  [665] = "-21.898000,-9.499000,118.777000,179.791000,0.392000,-123.893000,"
  [666] = "-21.901000,-9.495000,119.014000,179.790000,0.393000,-123.892000,"
  [667] = "-21.906000,-9.489000,119.373000,179.789000,0.396000,-123.892000,"
  [668] = "-21.912000,-9.481000,119.848000,179.788000,0.398000,-123.891000,"
  [669] = "-21.918000,-9.473000,120.297000,179.786000,0.401000,-123.890000,"
  [670] = "-21.923000,-9.467000,120.668000,179.785000,0.403000,-123.889000,"
  [671] = "-21.928000,-9.460000,121.039000,179.784000,0.406000,-123.888000,"
  [672] = "-21.845000,-9.093000,121.045000,179.788000,0.402000,-124.325000,"
  [673] = "-21.769000,-8.740000,121.052000,179.792000,0.397000,-124.728000,"
  [674] = "-21.697000,-8.391000,121.058000,179.797000,0.391000,-125.108000,"
  [675] = "-21.638000,-8.102000,121.063000,179.802000,0.385000,-125.409000,"
  [676] = "-21.575000,-7.782000,121.069000,179.807000,0.377000,-125.730000,"
  [677] = "-21.509000,-7.482000,121.076000,179.813000,0.367000,-126.051000,"
  [678] = "-21.413000,-7.146000,121.085000,179.824000,0.350000,-126.502000,"
  [679] = "-21.303000,-6.836000,121.095000,179.836000,0.330000,-127.021000,"
  [680] = "-21.191000,-6.564000,121.105000,179.848000,0.308000,-127.572000,"
  [681] = "-21.071000,-6.308000,121.115000,179.861000,0.286000,-128.189000,"
  [682] = "-20.932000,-6.069000,121.126000,179.875000,0.261000,-128.946000,"
  [683] = "-20.773000,-5.866000,121.138000,179.891000,0.232000,-129.864000,"
  [684] = "-20.590000,-5.697000,121.152000,179.909000,0.201000,-130.968000,"
  [685] = "-20.419000,-5.583000,121.164000,179.924000,0.172000,-132.053000,"
  [686] = "-20.230000,-5.492000,121.176000,179.939000,0.141000,-133.307000,"
  [687] = "-20.054000,-5.404000,121.187000,179.952000,0.115000,-134.556000,"
  [688] = "-19.877000,-5.305000,121.198000,179.963000,0.093000,-135.914000,"
  [689] = "-19.712000,-5.201000,121.207000,179.971000,0.074000,-137.273000,"
  [690] = "-19.569000,-5.104000,121.215000,179.977000,0.061000,-138.523000,"
  [691] = "-19.444000,-5.013000,121.222000,179.982000,0.050000,-139.689000,"
  [692] = "-19.298000,-4.901000,121.230000,179.986000,0.040000,-141.114000,"
  [693] = "-19.179000,-4.805000,121.236000,179.989000,0.033000,-142.336000,"
  [694] = "-19.074000,-4.717000,121.241000,179.991000,0.028000,-143.461000,"
  [695] = "-18.958000,-4.618000,121.246000,179.993000,0.023000,-144.749000,"
  [696] = "-18.847000,-4.521000,121.251000,179.994000,0.019000,-146.026000,"
  [697] = "-18.726000,-4.408000,121.257000,179.995000,0.015000,-147.486000,"
  [698] = "-18.617000,-4.297000,121.262000,179.996000,0.014000,-148.881000,"
  [699] = "-18.518000,-4.187000,121.266000,179.996000,0.014000,-150.220000,"
  [700] = "-18.428000,-4.079000,121.269000,179.996000,0.015000,-151.511000,"
  [701] = "-18.346000,-3.973000,121.272000,179.996000,0.018000,-152.759000,"
  [702] = "-18.250000,-3.838000,121.276000,179.995000,0.023000,-154.311000,"
  [703] = "-18.184000,-3.736000,121.278000,179.994000,0.029000,-155.473000,"
  [704] = "-18.124000,-3.635000,121.280000,179.993000,0.035000,-156.607000,"
  [705] = "-18.070000,-3.536000,121.281000,179.992000,0.042000,-157.716000,"
  [706] = "-17.998000,-3.393000,121.282000,179.990000,0.054000,-159.311000,"
  [707] = "-17.935000,-3.250000,121.283000,179.989000,0.068000,-160.916000,"
  [708] = "-17.880000,-3.116000,121.283000,179.987000,0.083000,-162.465000,"
  [709] = "-17.832000,-2.989000,121.283000,179.986000,0.099000,-163.999000,"
  [710] = "-17.789000,-2.868000,121.283000,179.985000,0.116000,-165.512000,"
  [711] = "-17.752000,-2.754000,121.282000,179.985000,0.134000,-167.010000,"
  [712] = "-17.720000,-2.646000,121.280000,179.985000,0.152000,-168.496000,"
  [713] = "-17.692000,-2.545000,121.279000,179.985000,0.171000,-169.972000,"
  [714] = "-17.668000,-2.449000,121.277000,179.986000,0.190000,-171.441000,"
  [715] = "-17.648000,-2.360000,121.275000,179.987000,0.210000,-172.903000,"
  [716] = "-17.631000,-2.277000,121.272000,179.989000,0.230000,-174.360000,"
  [717] = "-17.618000,-2.198000,121.269000,179.991000,0.251000,-175.808000,"
  [718] = "-17.612000,-2.118000,121.266000,179.993000,0.274000,-177.225000,"
  [719] = "-17.612000,-2.038000,121.262000,179.996000,0.298000,-178.614000,"
  [720] = "-17.621000,-1.930000,121.257000,-179.999000,0.331000,179.575000,"
  [721] = "-17.638000,-1.823000,121.250000,-179.993000,0.367000,177.803000,"
  [722] = "-17.664000,-1.717000,121.244000,-179.986000,0.404000,176.064000,"
  [723] = "-17.695000,-1.613000,121.236000,-179.978000,0.442000,174.351000,"
  [724] = "-17.729000,-1.512000,121.229000,-179.969000,0.479000,172.658000,"
  [725] = "-17.763000,-1.413000,121.222000,-179.959000,0.514000,170.982000,"
  [726] = "-17.796000,-1.317000,121.215000,-179.949000,0.547000,169.318000,"
  [727] = "-17.826000,-1.220000,121.209000,-179.938000,0.577000,167.683000,"
  [728] = "-17.857000,-1.115000,121.203000,-179.926000,0.605000,166.103000,"
  [729] = "-17.891000,-1.003000,121.197000,-179.914000,0.632000,164.577000,"
  [730] = "-17.927000,-0.883000,121.191000,-179.902000,0.658000,163.102000,"
  [731] = "-17.966000,-0.756000,121.185000,-179.890000,0.684000,161.676000,"
  [732] = "-18.010000,-0.622000,121.179000,-179.877000,0.710000,160.296000,"
  [733] = "-18.058000,-0.482000,121.172000,-179.863000,0.736000,158.960000,"
  [734] = "-18.112000,-0.336000,121.166000,-179.850000,0.762000,157.664000,"
  [735] = "-18.171000,-0.184000,121.159000,-179.835000,0.789000,156.408000,"
  [736] = "-18.236000,-0.028000,121.152000,-179.820000,0.817000,155.188000,"
  [737] = "-18.306000,0.130000,121.144000,-179.805000,0.846000,153.987000,"
  [738] = "-18.381000,0.285000,121.137000,-179.788000,0.875000,152.777000,"
  [739] = "-18.458000,0.435000,121.129000,-179.771000,0.903000,151.558000,"
  [740] = "-18.540000,0.581000,121.121000,-179.753000,0.932000,150.327000,"
  [741] = "-18.624000,0.723000,121.114000,-179.735000,0.959000,149.084000,"
  [742] = "-18.712000,0.860000,121.106000,-179.715000,0.987000,147.828000,"
  [743] = "-18.803000,0.992000,121.098000,-179.695000,1.014000,146.557000,"
  [744] = "-18.898000,1.119000,121.090000,-179.675000,1.040000,145.269000,"
  [745] = "-18.995000,1.242000,121.082000,-179.653000,1.066000,143.964000,"
  [746] = "-19.096000,1.359000,121.074000,-179.631000,1.091000,142.641000,"
  [747] = "-19.201000,1.474000,121.066000,-179.608000,1.116000,141.314000,"
  [748] = "-19.311000,1.597000,121.057000,-179.584000,1.143000,140.029000,"
  [749] = "-19.426000,1.728000,121.048000,-179.560000,1.171000,138.787000,"
  [750] = "-19.515000,1.831000,121.041000,-179.541000,1.193000,137.884000,"
  [751] = "-19.636000,1.977000,121.032000,-179.515000,1.222000,136.718000,"
  [752] = "-19.760000,2.132000,121.023000,-179.489000,1.252000,135.595000,"
  [753] = "-19.886000,2.297000,121.013000,-179.463000,1.282000,134.516000,"
  [754] = "-20.012000,2.472000,121.004000,-179.436000,1.312000,133.480000,"
  [755] = "-20.139000,2.659000,120.995000,-179.410000,1.341000,132.487000,"
  [756] = "-20.266000,2.856000,120.986000,-179.384000,1.369000,131.536000,"
  [757] = "-20.384000,3.053000,120.978000,-179.360000,1.394000,130.664000,"
  [758] = "-20.507000,3.265000,120.970000,-179.335000,1.418000,129.754000,"
  [759] = "-20.629000,3.481000,120.963000,-179.311000,1.440000,128.848000,"
  [760] = "-20.750000,3.700000,120.956000,-179.287000,1.460000,127.946000,"
  [761] = "-20.872000,3.924000,120.950000,-179.264000,1.478000,127.048000,"
  [762] = "-20.996000,4.150000,120.944000,-179.241000,1.495000,126.155000,"
  [763] = "-21.122000,4.379000,120.938000,-179.217000,1.512000,125.265000,"
  [764] = "-21.251000,4.611000,120.932000,-179.194000,1.528000,124.379000,"
  [765] = "-21.384000,4.845000,120.926000,-179.170000,1.544000,123.496000,"
  [766] = "-21.523000,5.081000,120.920000,-179.146000,1.560000,122.619000,"
  [767] = "-21.664000,5.325000,120.914000,-179.121000,1.579000,121.783000,"
  [768] = "-21.804000,5.576000,120.908000,-179.096000,1.598000,121.012000,"
  [769] = "-21.925000,5.801000,120.902000,-179.074000,1.616000,120.389000,"
  [770] = "-22.025000,5.996000,120.898000,-179.056000,1.632000,119.897000,"
  [771] = "-22.164000,6.281000,120.892000,-179.030000,1.654000,119.251000,"
  [772] = "-22.281000,6.538000,120.887000,-179.009000,1.674000,118.737000,"
  [773] = "-22.383000,6.779000,120.883000,-178.990000,1.691000,118.306000,"
  [774] = "-22.481000,7.031000,120.879000,-178.972000,1.708000,117.907000,"
  [775] = "-22.565000,7.263000,120.876000,-178.957000,1.722000,117.578000,"
  [776] = "-22.664000,7.566000,120.873000,-178.938000,1.739000,117.202000,"
  [777] = "-22.739000,7.817000,120.871000,-178.925000,1.752000,116.922000,"
  [778] = "-22.828000,8.137000,120.869000,-178.909000,1.765000,116.585000,"
  [779] = "-22.896000,8.399000,120.868000,-178.898000,1.775000,116.326000,"
  [780] = "-22.977000,8.733000,120.867000,-178.885000,1.785000,116.016000,"
  [781] = "-23.040000,9.006000,120.866000,-178.875000,1.793000,115.779000,"
  [782] = "-23.114000,9.353000,120.866000,-178.863000,1.801000,115.496000,"
  [783] = "-23.172000,9.636000,120.867000,-178.855000,1.807000,115.281000,"
  [784] = "-23.241000,9.995000,120.867000,-178.845000,1.814000,115.026000,"
  [785] = "-23.295000,10.287000,120.868000,-178.837000,1.820000,114.833000,"
  [786] = "-23.360000,10.657000,120.868000,-178.827000,1.827000,114.607000,"
  [787] = "-23.411000,10.956000,120.869000,-178.820000,1.832000,114.438000,"
  [788] = "-23.475000,11.334000,120.870000,-178.811000,1.840000,114.235000,"
  [789] = "-23.528000,11.637000,120.871000,-178.803000,1.846000,114.071000,"
  [790] = "-23.595000,12.015000,120.873000,-178.793000,1.853000,113.864000,"
  [791] = "-23.657000,12.356000,120.874000,-178.785000,1.859000,113.675000,"
  [792] = "-23.720000,12.697000,120.875000,-178.776000,1.866000,113.485000,"
  [793] = "-23.785000,13.039000,120.876000,-178.768000,1.872000,113.292000,"
  [794] = "-23.852000,13.381000,120.878000,-178.759000,1.878000,113.098000,"
  [795] = "-23.920000,13.723000,120.879000,-178.751000,1.884000,112.902000,"
  [796] = "-23.989000,14.066000,120.880000,-178.742000,1.890000,112.703000,"
  [797] = "-24.060000,14.410000,120.882000,-178.734000,1.895000,112.503000,"
  [798] = "-24.132000,14.754000,120.884000,-178.725000,1.901000,112.300000,"
  [799] = "-24.205000,15.098000,120.885000,-178.717000,1.906000,112.095000,"
  [800] = "-24.280000,15.443000,120.887000,-178.709000,1.910000,111.888000,"
  [801] = "-24.357000,15.789000,120.889000,-178.701000,1.915000,111.679000,"
  [802] = "-24.434000,16.135000,120.891000,-178.693000,1.919000,111.468000,"
  [803] = "-24.504000,16.444000,120.893000,-178.686000,1.922000,111.278000,"
  [804] = "-24.593000,16.831000,120.895000,-178.677000,1.926000,111.038000,"
  [805] = "-24.666000,17.141000,120.897000,-178.671000,1.929000,110.844000,"
  [806] = "-24.758000,17.529000,120.899000,-178.663000,1.931000,110.599000,"
  [807] = "-24.833000,17.841000,120.901000,-178.656000,1.933000,110.401000,"
  [808] = "-24.928000,18.232000,120.904000,-178.649000,1.935000,110.151000,"
  [809] = "-25.004000,18.546000,120.906000,-178.643000,1.936000,109.950000,"
  [810] = "-25.099000,18.941000,120.909000,-178.636000,1.937000,109.702000,"
  [811] = "-25.175000,19.259000,120.911000,-178.631000,1.938000,109.507000,"
  [812] = "-25.270000,19.660000,120.914000,-178.624000,1.938000,109.268000,"
  [813] = "-25.347000,19.982000,120.917000,-178.619000,1.939000,109.079000,"
  [814] = "-25.442000,20.388000,120.920000,-178.612000,1.940000,108.847000,"
  [815] = "-25.519000,20.713000,120.923000,-178.607000,1.941000,108.665000,"
  [816] = "-25.616000,21.122000,120.926000,-178.599000,1.943000,108.442000,"
  [817] = "-25.695000,21.451000,120.928000,-178.593000,1.945000,108.267000,"
  [818] = "-25.795000,21.863000,120.932000,-178.585000,1.949000,108.052000,"
  [819] = "-25.876000,22.194000,120.934000,-178.578000,1.953000,107.883000,"
  [820] = "-25.980000,22.607000,120.938000,-178.569000,1.957000,107.673000,"
  [821] = "-26.063000,22.939000,120.941000,-178.562000,1.961000,107.505000,"
  [822] = "-26.167000,23.357000,120.944000,-178.553000,1.966000,107.296000,"
  [823] = "-26.266000,23.765000,120.948000,-178.546000,1.968000,107.095000,"
  [824] = "-26.349000,24.120000,120.951000,-178.541000,1.969000,106.922000,"
  [825] = "-26.440000,24.538000,120.955000,-178.537000,1.967000,106.722000,"
  [826] = "-26.514000,24.903000,120.959000,-178.536000,1.962000,106.550000,"
  [827] = "-26.587000,25.305000,120.963000,-178.537000,1.954000,106.365000,"
  [828] = "-26.667000,25.705000,120.967000,-178.542000,1.940000,106.150000,"
  [829] = "-26.663000,25.706000,121.384000,-178.542000,1.941000,106.158000,"
  [830] = "-26.659000,25.708000,121.801000,-178.542000,1.941000,106.166000,"
  [831] = "-26.656000,25.710000,122.168000,-178.542000,1.941000,106.174000,"
  [832] = "-26.652000,25.711000,122.585000,-178.542000,1.941000,106.182000,"
  [833] = "-26.649000,25.713000,122.951000,-178.542000,1.941000,106.189000,"
  [834] = "-26.645000,25.714000,123.369000,-178.542000,1.941000,106.198000,"
  [835] = "-26.640000,25.716000,123.843000,-178.542000,1.941000,106.207000,"
  [836] = "-26.636000,25.718000,124.292000,-178.543000,1.942000,106.216000,"
  [837] = "-26.633000,25.719000,124.657000,-178.543000,1.942000,106.223000,"
  [838] = "-26.629000,25.721000,125.023000,-178.543000,1.942000,106.231000,"
  [839] = "-26.566000,25.344000,125.019000,-178.537000,1.956000,106.418000,"
  [840] = "-26.510000,24.896000,125.015000,-178.534000,1.966000,106.575000,"
  [841] = "-26.451000,24.520000,125.011000,-178.534000,1.970000,106.716000,"
  [842] = "-26.372000,24.093000,125.006000,-178.538000,1.972000,106.887000,"
  [843] = "-26.297000,23.732000,125.003000,-178.543000,1.971000,107.040000,"
  [844] = "-26.203000,23.321000,124.999000,-178.550000,1.967000,107.225000,"
  [845] = "-26.101000,22.902000,124.995000,-178.560000,1.962000,107.424000,"
  [846] = "-26.016000,22.570000,124.992000,-178.567000,1.957000,107.588000,"
  [847] = "-25.909000,22.159000,124.989000,-178.577000,1.951000,107.802000,"
  [848] = "-25.824000,21.831000,124.987000,-178.585000,1.947000,107.977000,"
  [849] = "-25.720000,21.422000,124.983000,-178.593000,1.944000,108.201000,"
  [850] = "-25.639000,21.096000,124.981000,-178.599000,1.942000,108.382000,"
  [851] = "-25.539000,20.688000,124.978000,-178.606000,1.940000,108.611000,"
  [852] = "-25.462000,20.363000,124.975000,-178.611000,1.939000,108.796000,"
  [853] = "-25.366000,19.958000,124.972000,-178.618000,1.939000,109.030000,"
  [854] = "-25.290000,19.635000,124.969000,-178.623000,1.939000,109.220000,"
  [855] = "-25.196000,19.234000,124.966000,-178.629000,1.939000,109.459000,"
  [856] = "-25.122000,18.914000,124.964000,-178.634000,1.938000,109.652000,"
  [857] = "-25.028000,18.518000,124.961000,-178.640000,1.938000,109.896000,"
  [858] = "-24.953000,18.202000,124.959000,-178.646000,1.937000,110.093000,"
  [859] = "-24.860000,17.810000,124.956000,-178.653000,1.936000,110.338000,"
  [860] = "-24.787000,17.497000,124.954000,-178.659000,1.934000,110.533000,"
  [861] = "-24.696000,17.107000,124.951000,-178.667000,1.931000,110.773000,"
  [862] = "-24.624000,16.796000,124.949000,-178.674000,1.928000,110.963000,"
  [863] = "-24.535000,16.409000,124.947000,-178.682000,1.924000,111.199000,"
  [864] = "-24.465000,16.100000,124.945000,-178.689000,1.921000,111.386000,"
  [865] = "-24.379000,15.714000,124.943000,-178.698000,1.916000,111.617000,"
  [866] = "-24.311000,15.407000,124.941000,-178.706000,1.912000,111.800000,"
  [867] = "-24.228000,15.023000,124.939000,-178.715000,1.906000,112.027000,"
  [868] = "-24.162000,14.717000,124.938000,-178.723000,1.901000,112.207000,"
  [869] = "-24.081000,14.335000,124.936000,-178.732000,1.895000,112.430000,"
  [870] = "-24.018000,14.030000,124.935000,-178.740000,1.890000,112.606000,"
  [871] = "-23.940000,13.649000,124.933000,-178.749000,1.883000,112.825000,"
  [872] = "-23.879000,13.345000,124.932000,-178.757000,1.878000,112.998000,"
  [873] = "-23.804000,12.965000,124.930000,-178.767000,1.871000,113.213000,"
  [874] = "-23.746000,12.662000,124.929000,-178.775000,1.865000,113.383000,"
  [875] = "-23.674000,12.283000,124.928000,-178.784000,1.858000,113.594000,"
  [876] = "-23.618000,11.980000,124.927000,-178.792000,1.852000,113.761000,"
  [877] = "-23.550000,11.602000,124.926000,-178.802000,1.844000,113.969000,"
  [878] = "-23.497000,11.300000,124.925000,-178.809000,1.838000,114.133000,"
  [879] = "-23.433000,10.923000,124.924000,-178.818000,1.831000,114.337000,"
  [880] = "-23.381000,10.623000,124.923000,-178.826000,1.826000,114.507000,"
  [881] = "-23.315000,10.253000,124.922000,-178.835000,1.819000,114.731000,"
  [882] = "-23.262000,9.960000,124.921000,-178.843000,1.813000,114.920000,"
  [883] = "-23.193000,9.599000,124.921000,-178.853000,1.806000,115.168000,"
  [884] = "-23.136000,9.315000,124.921000,-178.861000,1.800000,115.376000,"
  [885] = "-23.063000,8.965000,124.921000,-178.873000,1.792000,115.648000,"
  [886] = "-23.002000,8.689000,124.921000,-178.883000,1.784000,115.874000,"
  [887] = "-22.922000,8.351000,124.922000,-178.896000,1.773000,116.168000,"
  [888] = "-22.855000,8.085000,124.923000,-178.907000,1.763000,116.411000,"
  [889] = "-22.767000,7.760000,124.925000,-178.923000,1.749000,116.727000,"
  [890] = "-22.693000,7.505000,124.927000,-178.936000,1.736000,116.989000,"
  [891] = "-22.595000,7.198000,124.930000,-178.954000,1.718000,117.348000,"
  [892] = "-22.511000,6.963000,124.933000,-178.970000,1.703000,117.665000,"
  [893] = "-22.401000,6.681000,124.937000,-178.990000,1.685000,118.100000,"
  [894] = "-22.268000,6.370000,124.943000,-179.014000,1.662000,118.660000,"
  [895] = "-22.169000,6.158000,124.947000,-179.032000,1.646000,119.094000,"
  [896] = "-22.049000,5.914000,124.952000,-179.054000,1.627000,119.652000,"
  [897] = "-21.908000,5.644000,124.958000,-179.079000,1.606000,120.352000,"
  [898] = "-21.763000,5.382000,124.964000,-179.105000,1.586000,121.122000,"
  [899] = "-21.619000,5.133000,124.971000,-179.130000,1.567000,121.949000,"
  [900] = "-21.477000,4.896000,124.977000,-179.155000,1.550000,122.824000,"
  [901] = "-21.340000,4.662000,124.983000,-179.179000,1.534000,123.711000,"
  [902] = "-21.208000,4.430000,124.988000,-179.203000,1.518000,124.596000,"
  [903] = "-21.078000,4.199000,124.994000,-179.226000,1.502000,125.482000,"
  [904] = "-20.952000,3.971000,125.001000,-179.250000,1.485000,126.368000,"
  [905] = "-20.827000,3.745000,125.007000,-179.273000,1.466000,127.255000,"
  [906] = "-20.703000,3.521000,125.014000,-179.297000,1.446000,128.142000,"
  [907] = "-20.580000,3.301000,125.021000,-179.321000,1.424000,129.030000,"
  [908] = "-20.455000,3.084000,125.029000,-179.346000,1.400000,129.920000,"
  [909] = "-20.329000,2.870000,125.037000,-179.371000,1.374000,130.811000,"
  [910] = "-20.208000,2.676000,125.045000,-179.396000,1.347000,131.684000,"
  [911] = "-20.080000,2.483000,125.054000,-179.422000,1.318000,132.648000,"
  [912] = "-19.952000,2.301000,125.064000,-179.448000,1.289000,133.658000,"
  [913] = "-19.824000,2.131000,125.073000,-179.475000,1.259000,134.714000,"
  [914] = "-19.699000,1.972000,125.082000,-179.501000,1.230000,135.817000,"
  [915] = "-19.576000,1.822000,125.092000,-179.527000,1.200000,136.966000,"
  [916] = "-19.457000,1.682000,125.101000,-179.552000,1.172000,138.161000,"
  [917] = "-19.399000,1.616000,125.105000,-179.564000,1.158000,138.777000,"
  [918] = "-19.285000,1.490000,125.114000,-179.589000,1.131000,140.042000,"
  [919] = "-19.176000,1.373000,125.122000,-179.612000,1.106000,141.353000,"
  [920] = "-19.072000,1.259000,125.130000,-179.635000,1.081000,142.688000,"
  [921] = "-18.971000,1.141000,125.138000,-179.657000,1.055000,144.005000,"
  [922] = "-18.872000,1.018000,125.146000,-179.679000,1.029000,145.304000,"
  [923] = "-18.777000,0.889000,125.154000,-179.699000,1.002000,146.586000,"
  [924] = "-18.684000,0.756000,125.163000,-179.719000,0.974000,147.852000,"
  [925] = "-18.595000,0.619000,125.170000,-179.739000,0.946000,149.104000,"
  [926] = "-18.510000,0.477000,125.178000,-179.757000,0.918000,150.343000,"
  [927] = "-18.427000,0.330000,125.186000,-179.775000,0.889000,151.571000,"
  [928] = "-18.349000,0.180000,125.194000,-179.792000,0.861000,152.788000,"
  [929] = "-18.275000,0.026000,125.201000,-179.808000,0.832000,153.997000,"
  [930] = "-18.205000,-0.131000,125.209000,-179.823000,0.803000,155.207000,"
  [931] = "-18.142000,-0.284000,125.216000,-179.838000,0.776000,156.448000,"
  [932] = "-18.086000,-0.432000,125.222000,-179.852000,0.750000,157.723000,"
  [933] = "-18.034000,-0.574000,125.229000,-179.866000,0.724000,159.035000,"
  [934] = "-17.987000,-0.712000,125.235000,-179.879000,0.699000,160.385000,"
  [935] = "-17.945000,-0.843000,125.241000,-179.892000,0.674000,161.777000,"
  [936] = "-17.906000,-0.968000,125.247000,-179.904000,0.648000,163.212000,"
  [937] = "-17.869000,-1.087000,125.253000,-179.917000,0.621000,164.692000,"
  [938] = "-17.834000,-1.199000,125.259000,-179.928000,0.593000,166.221000,"
  [939] = "-17.800000,-1.304000,125.266000,-179.940000,0.564000,167.801000,"
  [940] = "-17.765000,-1.404000,125.272000,-179.951000,0.532000,169.423000,"
  [941] = "-17.727000,-1.504000,125.280000,-179.961000,0.497000,171.067000,"
  [942] = "-17.690000,-1.605000,125.287000,-179.971000,0.460000,172.733000,"
  [943] = "-17.655000,-1.707000,125.295000,-179.979000,0.422000,174.427000,"
  [944] = "-17.625000,-1.809000,125.302000,-179.987000,0.385000,176.153000,"
  [945] = "-17.604000,-1.911000,125.308000,-179.994000,0.349000,177.913000,"
  [946] = "-17.591000,-2.014000,125.314000,-179.999000,0.315000,179.710000,"
  [947] = "-17.588000,-2.116000,125.319000,179.996000,0.284000,-178.451000,"
  [948] = "-17.593000,-2.192000,125.322000,179.993000,0.261000,-177.039000,"
  [949] = "-17.604000,-2.267000,125.325000,179.991000,0.241000,-175.597000,"
  [950] = "-17.619000,-2.345000,125.328000,179.989000,0.221000,-174.138000,"
  [951] = "-17.638000,-2.428000,125.330000,179.987000,0.201000,-172.675000,"
  [952] = "-17.660000,-2.517000,125.332000,179.986000,0.182000,-171.208000,"
  [953] = "-17.686000,-2.612000,125.334000,179.985000,0.163000,-169.733000,"
  [954] = "-17.716000,-2.713000,125.335000,179.985000,0.145000,-168.250000,"
  [955] = "-17.750000,-2.820000,125.336000,179.985000,0.127000,-166.757000,"
  [956] = "-17.789000,-2.934000,125.337000,179.986000,0.110000,-165.250000,"
  [957] = "-17.833000,-3.054000,125.338000,179.987000,0.093000,-163.727000,"
  [958] = "-17.883000,-3.181000,125.338000,179.988000,0.078000,-162.184000,"
  [959] = "-17.940000,-3.312000,125.337000,179.989000,0.063000,-160.636000,"
  [960] = "-18.006000,-3.452000,125.337000,179.991000,0.050000,-159.018000,"
  [961] = "-18.081000,-3.589000,125.335000,179.992000,0.038000,-157.421000,"
  [962] = "-18.137000,-3.685000,125.333000,179.993000,0.032000,-156.307000,"
  [963] = "-18.199000,-3.782000,125.332000,179.994000,0.026000,-155.167000,"
  [964] = "-18.267000,-3.880000,125.329000,179.995000,0.022000,-153.999000,"
  [965] = "-18.365000,-4.010000,125.326000,179.996000,0.017000,-152.435000,"
  [966] = "-18.450000,-4.112000,125.323000,179.996000,0.015000,-151.181000,"
  [967] = "-18.542000,-4.216000,125.319000,179.996000,0.014000,-149.885000,"
  [968] = "-18.643000,-4.321000,125.315000,179.996000,0.014000,-148.540000,"
  [969] = "-18.755000,-4.427000,125.310000,179.995000,0.016000,-147.139000,"
  [970] = "-18.878000,-4.535000,125.304000,179.994000,0.020000,-145.674000,"
  [971] = "-19.010000,-4.645000,125.298000,179.992000,0.025000,-144.177000,"
  [972] = "-19.107000,-4.723000,125.294000,179.990000,0.030000,-143.115000,"
  [973] = "-19.218000,-4.808000,125.288000,179.987000,0.036000,-141.964000,"
  [974] = "-19.354000,-4.908000,125.281000,179.984000,0.046000,-140.605000,"
  [975] = "-19.499000,-5.005000,125.273000,179.979000,0.058000,-139.248000,"
  [976] = "-19.654000,-5.101000,125.265000,179.972000,0.073000,-137.874000,"
  [977] = "-19.807000,-5.186000,125.256000,179.964000,0.090000,-136.608000,"
  [978] = "-19.967000,-5.265000,125.247000,179.955000,0.110000,-135.363000,"
  [979] = "-20.149000,-5.343000,125.235000,179.942000,0.136000,-134.032000,"
  [980] = "-20.364000,-5.424000,125.222000,179.925000,0.170000,-132.579000,"
  [981] = "-20.532000,-5.511000,125.210000,179.911000,0.198000,-131.491000,"
  [982] = "-20.715000,-5.648000,125.197000,179.894000,0.229000,-130.351000,"
  [983] = "-20.882000,-5.823000,125.185000,179.878000,0.258000,-129.365000,"
  [984] = "-21.030000,-6.037000,125.173000,179.863000,0.285000,-128.524000,"
  [985] = "-21.152000,-6.267000,125.163000,179.850000,0.307000,-127.874000,"
  [986] = "-21.267000,-6.517000,125.153000,179.837000,0.328000,-127.293000,"
  [987] = "-21.382000,-6.815000,125.143000,179.825000,0.350000,-126.739000,"
  [988] = "-21.480000,-7.132000,125.134000,179.814000,0.367000,-126.276000,"
  [989] = "-21.543000,-7.396000,125.128000,179.807000,0.378000,-125.972000,"
  [990] = "-21.598000,-7.692000,125.122000,179.802000,0.385000,-125.695000,"
  [991] = "-21.665000,-8.058000,125.116000,179.797000,0.393000,-125.347000,"
  [992] = "-21.733000,-8.421000,125.109000,179.792000,0.399000,-124.984000,"
  [993] = "-21.787000,-8.696000,125.105000,179.789000,0.403000,-124.695000,"
  [994] = "-21.858000,-9.046000,125.099000,179.785000,0.407000,-124.311000,"
  [995] = "-21.936000,-9.408000,125.093000,179.782000,0.410000,-123.894000,"
  [996] = "-21.933000,-9.407000,125.510000,179.782000,0.408000,-123.892000,"
  [997] = "-21.930000,-9.405000,125.928000,179.783000,0.407000,-123.891000,"
  [998] = "-21.927000,-9.404000,126.295000,179.784000,0.405000,-123.890000,"
  [999] = "-21.924000,-9.403000,126.712000,179.785000,0.404000,-123.888000,"
  [1000] = "-21.921000,-9.402000,127.079000,179.785000,0.403000,-123.887000,"
  [1001] = "-21.918000,-9.401000,127.497000,179.786000,0.401000,-123.886000,"
  [1002] = "-21.914000,-9.399000,127.970000,179.787000,0.399000,-123.884000,"
  [1003] = "-21.911000,-9.398000,128.420000,179.788000,0.398000,-123.882000,"
  [1004] = "-21.908000,-9.397000,128.785000,179.789000,0.396000,-123.881000,"
  [1005] = "-21.905000,-9.396000,129.151000,179.789000,0.395000,-123.880000,"
  [1006] = "-21.841000,-9.094000,129.156000,179.792000,0.392000,-124.222000,"
  [1007] = "-21.767000,-8.722000,129.162000,179.796000,0.389000,-124.623000,"
  [1008] = "-21.698000,-8.350000,129.168000,179.800000,0.384000,-125.001000,"
  [1009] = "-21.636000,-7.996000,129.174000,179.804000,0.379000,-125.341000,"
  [1010] = "-21.574000,-7.627000,129.180000,179.808000,0.373000,-125.674000,"
  [1011] = "-21.527000,-7.331000,129.186000,179.812000,0.368000,-125.928000,"
  [1012] = "-21.474000,-7.055000,129.191000,179.817000,0.360000,-126.199000,"
  [1013] = "-21.387000,-6.733000,129.199000,179.826000,0.346000,-126.623000,"
  [1014] = "-21.274000,-6.415000,129.210000,179.838000,0.326000,-127.185000,"
  [1015] = "-21.178000,-6.199000,129.218000,179.848000,0.308000,-127.673000,"
  [1016] = "-21.058000,-5.968000,129.228000,179.861000,0.287000,-128.317000,"
  [1017] = "-20.945000,-5.787000,129.236000,179.872000,0.268000,-128.961000,"
  [1018] = "-20.800000,-5.610000,129.247000,179.886000,0.243000,-129.828000,"
  [1019] = "-20.652000,-5.478000,129.258000,179.900000,0.219000,-130.741000,"
  [1020] = "-20.476000,-5.365000,129.270000,179.915000,0.190000,-131.877000,"
  [1021] = "-20.289000,-5.287000,129.282000,179.931000,0.160000,-133.120000,"
  [1022] = "-20.088000,-5.227000,129.295000,179.946000,0.129000,-134.508000,"
  [1023] = "-19.895000,-5.156000,129.306000,179.959000,0.102000,-135.941000,"
  [1024] = "-19.715000,-5.077000,129.317000,179.969000,0.080000,-137.368000,"
  [1025] = "-19.561000,-4.999000,129.326000,179.976000,0.063000,-138.682000,"
  [1026] = "-19.427000,-4.922000,129.333000,179.982000,0.050000,-139.885000,"
  [1027] = "-19.274000,-4.826000,129.341000,179.987000,0.038000,-141.341000,"
  [1028] = "-19.151000,-4.740000,129.347000,179.990000,0.030000,-142.591000,"
  [1029] = "-19.043000,-4.661000,129.352000,179.992000,0.024000,-143.734000,"
  [1030] = "-18.902000,-4.550000,129.359000,179.994000,0.018000,-145.305000,"
  [1031] = "-18.775000,-4.444000,129.365000,179.996000,0.014000,-146.807000,"
  [1032] = "-18.658000,-4.341000,129.370000,179.997000,0.011000,-148.246000,"
  [1033] = "-18.553000,-4.238000,129.374000,179.997000,0.010000,-149.624000,"
  [1034] = "-18.457000,-4.137000,129.378000,179.997000,0.011000,-150.951000,"
  [1035] = "-18.370000,-4.037000,129.381000,179.997000,0.012000,-152.231000,"
  [1036] = "-18.290000,-3.938000,129.384000,179.996000,0.015000,-153.473000,"
  [1037] = "-18.217000,-3.841000,129.387000,179.996000,0.020000,-154.679000,"
  [1038] = "-18.151000,-3.745000,129.389000,179.995000,0.025000,-155.853000,"
  [1039] = "-18.090000,-3.651000,129.390000,179.994000,0.031000,-157.000000,"
  [1040] = "-18.035000,-3.558000,129.392000,179.993000,0.038000,-158.121000,"
  [1041] = "-17.962000,-3.424000,129.393000,179.991000,0.049000,-159.732000,"
  [1042] = "-17.898000,-3.289000,129.394000,179.990000,0.063000,-161.357000,"
  [1043] = "-17.843000,-3.162000,129.394000,179.988000,0.078000,-162.916000,"
  [1044] = "-17.795000,-3.040000,129.394000,179.987000,0.094000,-164.461000,"
  [1045] = "-17.752000,-2.925000,129.393000,179.986000,0.111000,-165.983000,"
  [1046] = "-17.715000,-2.816000,129.392000,179.986000,0.128000,-167.488000,"
  [1047] = "-17.683000,-2.713000,129.391000,179.986000,0.146000,-168.981000,"
  [1048] = "-17.654000,-2.616000,129.389000,179.986000,0.164000,-170.464000,"
  [1049] = "-17.630000,-2.525000,129.388000,179.987000,0.183000,-171.939000,"
  [1050] = "-17.608000,-2.440000,129.386000,179.988000,0.202000,-173.407000,"
  [1051] = "-17.590000,-2.360000,129.383000,179.990000,0.221000,-174.871000,"
  [1052] = "-17.574000,-2.286000,129.381000,179.992000,0.241000,-176.331000,"
  [1053] = "-17.563000,-2.215000,129.378000,179.995000,0.261000,-177.777000,"
  [1054] = "-17.557000,-2.118000,129.374000,179.999000,0.290000,-179.658000,"
  [1055] = "-17.561000,-2.020000,129.368000,-179.996000,0.321000,178.508000,"
  [1056] = "-17.575000,-1.922000,129.363000,-179.990000,0.354000,176.715000,"
  [1057] = "-17.597000,-1.824000,129.356000,-179.983000,0.389000,174.957000,"
  [1058] = "-17.628000,-1.725000,129.349000,-179.975000,0.426000,173.239000,"
  [1059] = "-17.665000,-1.624000,129.342000,-179.966000,0.463000,171.562000,"
  [1060] = "-17.705000,-1.521000,129.334000,-179.956000,0.500000,169.920000,"
  [1061] = "-17.745000,-1.417000,129.327000,-179.945000,0.534000,168.309000,"
  [1062] = "-17.784000,-1.312000,129.320000,-179.934000,0.566000,166.727000,"
  [1063] = "-17.822000,-1.201000,129.313000,-179.923000,0.596000,165.189000,"
  [1064] = "-17.860000,-1.084000,129.307000,-179.911000,0.624000,163.696000,"
  [1065] = "-17.899000,-0.961000,129.301000,-179.898000,0.651000,162.246000,"
  [1066] = "-17.941000,-0.832000,129.295000,-179.886000,0.676000,160.836000,"
  [1067] = "-17.986000,-0.698000,129.289000,-179.873000,0.702000,159.465000,"
  [1068] = "-18.036000,-0.559000,129.283000,-179.860000,0.727000,158.130000,"
  [1069] = "-18.090000,-0.416000,129.276000,-179.846000,0.752000,156.830000,"
  [1070] = "-18.150000,-0.268000,129.269000,-179.831000,0.779000,155.562000,"
  [1071] = "-18.216000,-0.116000,129.262000,-179.816000,0.806000,154.324000,"
  [1072] = "-18.289000,0.038000,129.255000,-179.800000,0.835000,153.111000,"
  [1073] = "-18.367000,0.189000,129.247000,-179.784000,0.864000,151.895000,"
  [1074] = "-18.450000,0.336000,129.239000,-179.766000,0.893000,150.671000,"
  [1075] = "-18.536000,0.479000,129.231000,-179.748000,0.922000,149.437000,"
  [1076] = "-18.626000,0.618000,129.223000,-179.729000,0.951000,148.192000,"
  [1077] = "-18.720000,0.753000,129.215000,-179.709000,0.980000,146.934000,"
  [1078] = "-18.817000,0.883000,129.206000,-179.688000,1.008000,145.662000,"
  [1079] = "-18.916000,1.008000,129.198000,-179.667000,1.036000,144.375000,"
  [1080] = "-19.018000,1.129000,129.190000,-179.645000,1.062000,143.071000,"
  [1081] = "-19.123000,1.245000,129.182000,-179.623000,1.088000,141.749000,"
  [1082] = "-19.230000,1.357000,129.174000,-179.599000,1.113000,140.412000,"
  [1083] = "-19.341000,1.476000,129.165000,-179.575000,1.139000,139.111000,"
  [1084] = "-19.398000,1.539000,129.161000,-179.563000,1.152000,138.478000,"
  [1085] = "-19.486000,1.638000,129.154000,-179.545000,1.172000,137.552000,"
  [1086] = "-19.606000,1.778000,129.145000,-179.519000,1.200000,136.360000,"
  [1087] = "-19.729000,1.929000,129.136000,-179.494000,1.229000,135.217000,"
  [1088] = "-19.855000,2.090000,129.127000,-179.468000,1.258000,134.123000,"
  [1089] = "-19.983000,2.263000,129.118000,-179.441000,1.287000,133.079000,"
  [1090] = "-20.112000,2.448000,129.108000,-179.415000,1.316000,132.083000,"
  [1091] = "-20.242000,2.645000,129.099000,-179.389000,1.345000,131.137000,"
  [1092] = "-20.371000,2.854000,129.090000,-179.363000,1.374000,130.240000,"
  [1093] = "-20.499000,3.072000,129.082000,-179.337000,1.401000,129.370000,"
  [1094] = "-20.626000,3.293000,129.074000,-179.313000,1.425000,128.499000,"
  [1095] = "-20.752000,3.517000,129.067000,-179.288000,1.448000,127.626000,"
  [1096] = "-20.879000,3.742000,129.060000,-179.264000,1.468000,126.751000,"
  [1097] = "-21.007000,3.970000,129.053000,-179.240000,1.487000,125.875000,"
  [1098] = "-21.136000,4.200000,129.047000,-179.216000,1.505000,124.995000,"
  [1099] = "-21.268000,4.431000,129.041000,-179.193000,1.522000,124.113000,"
  [1100] = "-21.403000,4.663000,129.035000,-179.169000,1.538000,123.227000,"
  [1101] = "-21.507000,4.838000,129.031000,-179.151000,1.550000,122.561000,"
  [1102] = "-21.643000,5.061000,129.025000,-179.127000,1.566000,121.720000,"
  [1103] = "-21.788000,5.308000,129.019000,-179.102000,1.583000,120.881000,"
  [1104] = "-21.934000,5.568000,129.013000,-179.076000,1.603000,120.103000,"
  [1105] = "-22.076000,5.838000,129.007000,-179.051000,1.623000,119.399000,"
  [1106] = "-22.196000,6.082000,129.002000,-179.030000,1.642000,118.842000,"
  [1107] = "-22.294000,6.295000,128.998000,-179.012000,1.657000,118.410000,"
  [1108] = "-22.427000,6.609000,128.993000,-178.988000,1.679000,117.857000,"
  [1109] = "-22.536000,6.893000,128.989000,-178.968000,1.698000,117.431000,"
  [1110] = "-22.629000,7.161000,128.985000,-178.951000,1.714000,117.087000,"
  [1111] = "-22.717000,7.442000,128.983000,-178.935000,1.730000,116.780000,"
  [1112] = "-22.789000,7.701000,128.981000,-178.922000,1.743000,116.535000,"
  [1113] = "-22.875000,8.032000,128.979000,-178.907000,1.758000,116.241000,"
  [1114] = "-22.941000,8.301000,128.978000,-178.895000,1.768000,116.012000,"
  [1115] = "-23.019000,8.644000,128.977000,-178.882000,1.780000,115.735000,"
  [1116] = "-23.079000,8.922000,128.976000,-178.873000,1.787000,115.520000,"
  [1117] = "-23.152000,9.275000,128.976000,-178.861000,1.796000,115.261000,"
  [1118] = "-23.214000,9.597000,128.977000,-178.852000,1.803000,115.036000,"
  [1119] = "-23.276000,9.924000,128.977000,-178.843000,1.810000,114.819000,"
  [1120] = "-23.329000,10.217000,128.978000,-178.835000,1.815000,114.634000,"
  [1121] = "-23.395000,10.588000,128.979000,-178.826000,1.822000,114.411000,"
  [1122] = "-23.446000,10.887000,128.980000,-178.819000,1.827000,114.240000,"
  [1123] = "-23.512000,11.264000,128.981000,-178.810000,1.834000,114.035000,"
  [1124] = "-23.565000,11.566000,128.982000,-178.802000,1.840000,113.870000,"
  [1125] = "-23.634000,11.944000,128.983000,-178.792000,1.847000,113.662000,"
  [1126] = "-23.698000,12.284000,128.984000,-178.784000,1.854000,113.474000,"
  [1127] = "-23.763000,12.625000,128.985000,-178.775000,1.861000,113.284000,"
  [1128] = "-23.822000,12.928000,128.986000,-178.767000,1.866000,113.114000,"
  [1129] = "-23.897000,13.307000,128.988000,-178.757000,1.874000,112.900000,"
  [1130] = "-23.959000,13.611000,128.989000,-178.750000,1.879000,112.728000,"
  [1131] = "-24.038000,13.992000,128.990000,-178.740000,1.886000,112.511000,"
  [1132] = "-24.102000,14.297000,128.992000,-178.732000,1.892000,112.336000,"
  [1133] = "-24.183000,14.679000,128.994000,-178.722000,1.898000,112.116000,"
  [1134] = "-24.257000,15.023000,128.995000,-178.714000,1.904000,111.916000,"
  [1135] = "-24.333000,15.369000,128.997000,-178.705000,1.909000,111.714000,"
  [1136] = "-24.401000,15.677000,128.999000,-178.698000,1.913000,111.534000,"
  [1137] = "-24.487000,16.063000,129.001000,-178.689000,1.919000,111.306000,"
  [1138] = "-24.556000,16.372000,129.002000,-178.682000,1.922000,111.123000,"
  [1139] = "-24.644000,16.761000,129.005000,-178.673000,1.926000,110.892000,"
  [1140] = "-24.715000,17.073000,129.007000,-178.667000,1.929000,110.705000,"
  [1141] = "-24.805000,17.464000,129.009000,-178.659000,1.932000,110.470000,"
  [1142] = "-24.887000,17.817000,129.012000,-178.652000,1.934000,110.257000,"
  [1143] = "-24.969000,18.172000,129.014000,-178.646000,1.936000,110.042000,"
  [1144] = "-25.042000,18.489000,129.017000,-178.640000,1.936000,109.850000,"
  [1145] = "-25.134000,18.887000,129.020000,-178.634000,1.937000,109.610000,"
  [1146] = "-25.207000,19.207000,129.022000,-178.629000,1.937000,109.419000,"
  [1147] = "-25.300000,19.609000,129.025000,-178.623000,1.936000,109.180000,"
  [1148] = "-25.376000,19.932000,129.028000,-178.619000,1.936000,108.990000,"
  [1149] = "-25.472000,20.336000,129.031000,-178.613000,1.936000,108.752000,"
  [1150] = "-25.562000,20.701000,129.034000,-178.607000,1.937000,108.540000,"
  [1151] = "-25.653000,21.066000,129.037000,-178.600000,1.938000,108.327000,"
  [1152] = "-25.737000,21.390000,129.039000,-178.594000,1.940000,108.139000,"
  [1153] = "-25.846000,21.795000,129.042000,-178.586000,1.943000,107.904000,"
  [1154] = "-25.936000,22.119000,129.045000,-178.578000,1.947000,107.719000,"
  [1155] = "-26.047000,22.528000,129.048000,-178.568000,1.953000,107.502000,"
  [1156] = "-26.133000,22.859000,129.051000,-178.559000,1.959000,107.339000,"
  [1157] = "-26.233000,23.280000,129.054000,-178.550000,1.965000,107.151000,"
  [1158] = "-26.315000,23.667000,129.058000,-178.543000,1.969000,106.995000,"
  [1159] = "-26.388000,24.063000,129.062000,-178.537000,1.972000,106.853000,"
  [1160] = "-26.452000,24.500000,129.067000,-178.534000,1.971000,106.716000,"
  [1161] = "-26.494000,24.888000,129.071000,-178.534000,1.967000,106.610000,"
  [1162] = "-26.526000,25.353000,129.077000,-178.539000,1.957000,106.502000,"
  [1163] = "-26.572000,25.741000,129.081000,-178.546000,1.942000,106.344000,"
  [1164] = "-26.564000,25.744000,129.498000,-178.546000,1.941000,106.357000,"
  [1165] = "-26.557000,25.747000,129.915000,-178.547000,1.941000,106.370000,"
  [1166] = "-26.549000,25.750000,130.379000,-178.548000,1.941000,106.384000,"
  [1167] = "-26.544000,25.753000,130.721000,-178.548000,1.941000,106.395000,"
  [1168] = "-26.538000,25.755000,131.062000,-178.548000,1.940000,106.405000,"
  [1169] = "-26.530000,25.758000,131.484000,-178.549000,1.940000,106.418000,"
  [1170] = "-26.522000,25.761000,131.958000,-178.550000,1.940000,106.433000,"
  [1171] = "-26.515000,25.765000,132.407000,-178.550000,1.940000,106.447000,"
  [1172] = "-26.508000,25.767000,132.773000,-178.551000,1.939000,106.458000,"
  [1173] = "-26.502000,25.770000,133.139000,-178.551000,1.939000,106.470000,"
  [1174] = "-26.473000,25.370000,133.135000,-178.543000,1.955000,106.597000,"
  [1175] = "-26.468000,24.887000,133.129000,-178.537000,1.964000,106.651000,"
  [1176] = "-26.444000,24.487000,133.124000,-178.536000,1.968000,106.718000,"
  [1177] = "-26.396000,24.038000,133.119000,-178.539000,1.968000,106.819000,"
  [1178] = "-26.339000,23.664000,133.114000,-178.544000,1.965000,106.926000,"
  [1179] = "-26.258000,23.242000,133.110000,-178.552000,1.960000,107.072000,"
  [1180] = "-26.160000,22.819000,133.107000,-178.561000,1.953000,107.250000,"
  [1181] = "-26.074000,22.488000,133.104000,-178.570000,1.947000,107.410000,"
  [1182] = "-25.959000,22.082000,133.101000,-178.580000,1.941000,107.634000,"
  [1183] = "-25.864000,21.762000,133.099000,-178.588000,1.937000,107.830000,"
  [1184] = "-25.749000,21.362000,133.096000,-178.597000,1.933000,108.077000,"
  [1185] = "-25.662000,21.040000,133.093000,-178.603000,1.932000,108.273000,"
  [1186] = "-25.557000,20.637000,133.090000,-178.610000,1.931000,108.517000,"
  [1187] = "-25.476000,20.315000,133.088000,-178.616000,1.930000,108.711000,"
  [1188] = "-25.379000,19.911000,133.085000,-178.622000,1.931000,108.952000,"
  [1189] = "-25.303000,19.589000,133.082000,-178.626000,1.931000,109.143000,"
  [1190] = "-25.210000,19.187000,133.079000,-178.632000,1.931000,109.381000,"
  [1191] = "-25.137000,18.866000,133.076000,-178.637000,1.931000,109.570000,"
  [1192] = "-25.047000,18.466000,133.073000,-178.643000,1.931000,109.805000,"
  [1193] = "-24.975000,18.148000,133.071000,-178.648000,1.930000,109.992000,"
  [1194] = "-24.886000,17.752000,133.068000,-178.655000,1.929000,110.224000,"
  [1195] = "-24.815000,17.437000,133.066000,-178.661000,1.927000,110.408000,"
  [1196] = "-24.727000,17.044000,133.063000,-178.669000,1.924000,110.637000,"
  [1197] = "-24.656000,16.732000,133.061000,-178.676000,1.921000,110.819000,"
  [1198] = "-24.569000,16.342000,133.059000,-178.684000,1.916000,111.045000,"
  [1199] = "-24.499000,16.032000,133.057000,-178.691000,1.912000,111.225000,"
  [1200] = "-24.414000,15.645000,133.055000,-178.700000,1.907000,111.449000,"
  [1201] = "-24.346000,15.337000,133.053000,-178.708000,1.902000,111.626000,"
  [1202] = "-24.262000,14.953000,133.052000,-178.717000,1.896000,111.847000,"
  [1203] = "-24.196000,14.646000,133.050000,-178.725000,1.891000,112.023000,"
  [1204] = "-24.114000,14.264000,133.048000,-178.734000,1.885000,112.241000,"
  [1205] = "-24.050000,13.959000,133.047000,-178.742000,1.879000,112.414000,"
  [1206] = "-23.971000,13.578000,133.046000,-178.752000,1.872000,112.630000,"
  [1207] = "-23.909000,13.274000,133.044000,-178.760000,1.866000,112.801000,"
  [1208] = "-23.833000,12.895000,133.043000,-178.770000,1.859000,113.015000,"
  [1209] = "-23.773000,12.592000,133.042000,-178.778000,1.853000,113.184000,"
  [1210] = "-23.700000,12.214000,133.041000,-178.787000,1.846000,113.395000,"
  [1211] = "-23.643000,11.912000,133.040000,-178.795000,1.840000,113.563000,"
  [1212] = "-23.574000,11.535000,133.038000,-178.804000,1.833000,113.772000,"
  [1213] = "-23.520000,11.233000,133.038000,-178.812000,1.827000,113.938000,"
  [1214] = "-23.454000,10.857000,133.036000,-178.821000,1.821000,114.145000,"
  [1215] = "-23.401000,10.558000,133.036000,-178.828000,1.815000,114.316000,"
  [1216] = "-23.336000,10.187000,133.035000,-178.837000,1.809000,114.537000,"
  [1217] = "-23.283000,9.892000,133.034000,-178.845000,1.803000,114.719000,"
  [1218] = "-23.216000,9.528000,133.033000,-178.855000,1.796000,114.953000,"
  [1219] = "-23.161000,9.240000,133.033000,-178.863000,1.790000,115.146000,"
  [1220] = "-23.090000,8.884000,133.033000,-178.874000,1.781000,115.394000,"
  [1221] = "-23.031000,8.602000,133.033000,-178.883000,1.773000,115.597000,"
  [1222] = "-22.955000,8.255000,133.034000,-178.896000,1.762000,115.857000,"
  [1223] = "-22.891000,7.982000,133.035000,-178.907000,1.751000,116.070000,"
  [1224] = "-22.807000,7.645000,133.037000,-178.922000,1.736000,116.343000,"
  [1225] = "-22.736000,7.382000,133.039000,-178.935000,1.723000,116.573000,"
  [1226] = "-22.640000,7.067000,133.042000,-178.953000,1.706000,116.902000,"
  [1227] = "-22.558000,6.827000,133.044000,-178.968000,1.691000,117.201000,"
  [1228] = "-22.462000,6.568000,133.048000,-178.985000,1.675000,117.574000,"
  [1229] = "-22.361000,6.321000,133.052000,-179.003000,1.659000,117.987000,"
  [1230] = "-22.245000,6.060000,133.056000,-179.024000,1.641000,118.489000,"
  [1231] = "-22.106000,5.772000,133.062000,-179.048000,1.621000,119.134000,"
  [1232] = "-22.005000,5.577000,133.066000,-179.065000,1.607000,119.631000,"
  [1233] = "-21.884000,5.355000,133.071000,-179.087000,1.591000,120.269000,"
  [1234] = "-21.741000,5.109000,133.077000,-179.111000,1.573000,121.067000,"
  [1235] = "-21.604000,4.885000,133.082000,-179.135000,1.558000,121.894000,"
  [1236] = "-21.497000,4.710000,133.087000,-179.153000,1.546000,122.563000,"
  [1237] = "-21.358000,4.477000,133.093000,-179.177000,1.529000,123.448000,"
  [1238] = "-21.222000,4.246000,133.099000,-179.201000,1.512000,124.328000,"
  [1239] = "-21.089000,4.015000,133.105000,-179.226000,1.494000,125.202000,"
  [1240] = "-20.958000,3.785000,133.112000,-179.250000,1.474000,126.070000,"
  [1241] = "-20.827000,3.558000,133.119000,-179.274000,1.453000,126.934000,"
  [1242] = "-20.698000,3.331000,133.127000,-179.299000,1.430000,127.794000,"
  [1243] = "-20.568000,3.107000,133.134000,-179.324000,1.405000,128.650000,"
  [1244] = "-20.438000,2.885000,133.143000,-179.350000,1.378000,129.501000,"
  [1245] = "-20.307000,2.668000,133.151000,-179.376000,1.350000,130.368000,"
  [1246] = "-20.176000,2.465000,133.160000,-179.402000,1.321000,131.285000,"
  [1247] = "-20.046000,2.274000,133.170000,-179.428000,1.292000,132.254000,"
  [1248] = "-19.917000,2.095000,133.179000,-179.454000,1.263000,133.274000,"
  [1249] = "-19.790000,1.928000,133.188000,-179.480000,1.235000,134.346000,"
  [1250] = "-19.665000,1.773000,133.197000,-179.506000,1.207000,135.469000,"
  [1251] = "-19.544000,1.629000,133.206000,-179.531000,1.179000,136.643000,"
  [1252] = "-19.426000,1.495000,133.215000,-179.556000,1.152000,137.868000,"
  [1253] = "-19.311000,1.372000,133.223000,-179.580000,1.126000,139.143000,"
  [1254] = "-19.201000,1.258000,133.232000,-179.604000,1.101000,140.467000,"
  [1255] = "-19.092000,1.145000,133.240000,-179.627000,1.076000,141.797000,"
  [1256] = "-18.986000,1.027000,133.248000,-179.650000,1.049000,143.108000,"
  [1257] = "-18.881000,0.905000,133.257000,-179.672000,1.021000,144.403000,"
  [1258] = "-18.779000,0.779000,133.265000,-179.694000,0.992000,145.683000,"
  [1259] = "-18.679000,0.649000,133.274000,-179.714000,0.962000,146.949000,"
  [1260] = "-18.583000,0.514000,133.282000,-179.734000,0.933000,148.203000,"
  [1261] = "-18.490000,0.376000,133.291000,-179.754000,0.902000,149.446000,"
  [1262] = "-18.401000,0.233000,133.299000,-179.772000,0.872000,150.680000,"
  [1263] = "-18.317000,0.087000,133.307000,-179.789000,0.842000,151.906000,"
  [1264] = "-18.238000,-0.063000,133.315000,-179.806000,0.813000,153.125000,"
  [1265] = "-18.165000,-0.214000,133.322000,-179.822000,0.784000,154.356000,"
  [1266] = "-18.100000,-0.361000,133.329000,-179.836000,0.757000,155.614000,"
  [1267] = "-18.040000,-0.506000,133.336000,-179.851000,0.731000,156.898000,"
  [1268] = "-17.986000,-0.647000,133.343000,-179.864000,0.705000,158.212000,"
  [1269] = "-17.937000,-0.784000,133.349000,-179.877000,0.680000,159.558000,"
  [1270] = "-17.891000,-0.916000,133.355000,-179.890000,0.654000,160.936000,"
  [1271] = "-17.847000,-1.044000,133.361000,-179.903000,0.627000,162.349000,"
  [1272] = "-17.806000,-1.167000,133.368000,-179.915000,0.600000,163.800000,"
  [1273] = "-17.765000,-1.285000,133.374000,-179.926000,0.571000,165.289000,"
  [1274] = "-17.724000,-1.398000,133.381000,-179.938000,0.539000,166.819000,"
  [1275] = "-17.681000,-1.507000,133.388000,-179.949000,0.506000,168.386000,"
  [1276] = "-17.639000,-1.613000,133.396000,-179.959000,0.470000,169.990000,"
  [1277] = "-17.600000,-1.716000,133.403000,-179.968000,0.434000,171.637000,"
  [1278] = "-17.567000,-1.814000,133.410000,-179.977000,0.398000,173.330000,"
  [1279] = "-17.542000,-1.909000,133.417000,-179.984000,0.364000,175.074000,"
  [1280] = "-17.526000,-2.004000,133.423000,-179.991000,0.331000,176.854000,"
  [1281] = "-17.519000,-2.098000,133.428000,-179.997000,0.300000,178.672000,"
  [1282] = "-17.521000,-2.191000,133.433000,179.999000,0.271000,-179.467000,"
  [1283] = "-17.533000,-2.282000,133.436000,179.995000,0.244000,-177.556000,"
  [1284] = "-17.547000,-2.352000,133.439000,179.992000,0.225000,-176.097000,"
  [1285] = "-17.564000,-2.427000,133.441000,179.990000,0.206000,-174.634000,"
  [1286] = "-17.584000,-2.507000,133.444000,179.989000,0.187000,-173.168000,"
  [1287] = "-17.606000,-2.592000,133.446000,179.988000,0.168000,-171.696000,"
  [1288] = "-17.632000,-2.683000,133.447000,179.987000,0.149000,-170.217000,"
  [1289] = "-17.662000,-2.781000,133.449000,179.987000,0.131000,-168.728000,"
  [1290] = "-17.695000,-2.884000,133.450000,179.987000,0.114000,-167.229000,"
  [1291] = "-17.734000,-2.992000,133.451000,179.988000,0.096000,-165.715000,"
  [1292] = "-17.778000,-3.107000,133.451000,179.989000,0.080000,-164.183000,"
  [1293] = "-17.828000,-3.228000,133.452000,179.990000,0.065000,-162.630000,"
  [1294] = "-17.885000,-3.352000,133.451000,179.992000,0.050000,-161.071000,"
  [1295] = "-17.941000,-3.460000,133.450000,179.993000,0.039000,-159.719000,"
  [1296] = "-18.004000,-3.572000,133.449000,179.994000,0.030000,-158.326000,"
  [1297] = "-18.086000,-3.702000,133.447000,179.996000,0.020000,-156.692000,"
  [1298] = "-18.149000,-3.793000,133.445000,179.997000,0.015000,-155.540000,"
  [1299] = "-18.239000,-3.912000,133.442000,179.998000,0.009000,-154.009000,"
  [1300] = "-18.340000,-4.035000,133.439000,179.999000,0.005000,-152.408000,"
  [1301] = "-18.428000,-4.132000,133.435000,179.999000,0.003000,-151.121000,"
  [1302] = "-18.524000,-4.230000,133.432000,179.999000,0.003000,-149.790000,"
  [1303] = "-18.629000,-4.329000,133.427000,179.999000,0.003000,-148.406000,"
  [1304] = "-18.745000,-4.429000,133.422000,179.998000,0.006000,-146.962000,"
  [1305] = "-18.872000,-4.532000,133.417000,179.997000,0.010000,-145.455000,"
  [1306] = "-19.013000,-4.638000,133.410000,179.995000,0.016000,-143.875000,"
  [1307] = "-19.139000,-4.724000,133.404000,179.992000,0.023000,-142.545000,"
  [1308] = "-19.271000,-4.808000,133.397000,179.989000,0.032000,-141.215000,"
  [1309] = "-19.406000,-4.884000,133.390000,179.984000,0.043000,-139.934000,"
  [1310] = "-19.568000,-4.965000,133.382000,179.978000,0.059000,-138.494000,"
  [1311] = "-19.744000,-5.039000,133.372000,179.969000,0.079000,-137.025000,"
  [1312] = "-19.888000,-5.091000,133.364000,179.961000,0.097000,-135.888000,"
  [1313] = "-20.084000,-5.149000,133.352000,179.948000,0.124000,-134.438000,"
  [1314] = "-20.260000,-5.193000,133.341000,179.935000,0.151000,-133.204000,"
  [1315] = "-20.439000,-5.265000,133.330000,179.921000,0.178000,-131.980000,"
  [1316] = "-20.607000,-5.369000,133.318000,179.907000,0.204000,-130.856000,"
  [1317] = "-20.778000,-5.525000,133.306000,179.892000,0.231000,-129.751000,"
  [1318] = "-20.919000,-5.704000,133.296000,179.879000,0.253000,-128.881000,"
  [1319] = "-21.060000,-5.945000,133.285000,179.866000,0.275000,-128.052000,"
  [1320] = "-21.152000,-6.136000,133.277000,179.857000,0.291000,-127.539000,"
  [1321] = "-21.259000,-6.406000,133.268000,179.846000,0.308000,-126.971000,"
  [1322] = "-21.345000,-6.690000,133.260000,179.838000,0.322000,-126.521000,"
  [1323] = "-21.423000,-7.060000,133.252000,179.831000,0.333000,-126.105000,"
  [1324] = "-21.466000,-7.358000,133.247000,179.828000,0.337000,-125.860000,"
  [1325] = "-21.508000,-7.649000,133.243000,179.825000,0.341000,-125.618000,"
  [1326] = "-21.565000,-8.012000,133.237000,179.821000,0.346000,-125.296000,"
  [1327] = "-21.629000,-8.388000,133.231000,179.818000,0.350000,-124.942000,"
  [1328] = "-21.681000,-8.672000,133.226000,179.815000,0.354000,-124.658000,"
  [1329] = "-21.752000,-9.030000,133.220000,179.811000,0.358000,-124.281000,"
  [1330] = "-21.827000,-9.376000,133.214000,179.807000,0.362000,-123.894000,"
  [1331] = "-21.815000,-9.377000,133.632000,179.810000,0.357000,-123.893000,"
  [1332] = "-21.804000,-9.377000,134.050000,179.813000,0.352000,-123.892000,"
  [1333] = "-21.791000,-9.378000,134.514000,179.816000,0.346000,-123.891000,"
  [1334] = "-21.781000,-9.378000,134.858000,179.818000,0.342000,-123.890000,"
  [1335] = "-21.771000,-9.379000,135.201000,179.820000,0.337000,-123.889000,"
  [1336] = "-21.759000,-9.379000,135.622000,179.823000,0.332000,-123.888000,"
  [1337] = "-21.745000,-9.380000,136.110000,179.826000,0.326000,-123.887000,"
  [1338] = "-21.731000,-9.381000,136.566000,179.829000,0.321000,-123.886000,"
  [1339] = "-21.720000,-9.382000,136.955000,179.832000,0.316000,-123.885000,"
  [1340] = "-21.708000,-9.383000,137.344000,179.834000,0.311000,-123.885000,"
  [1341] = "-21.638000,-9.082000,137.350000,179.838000,0.306000,-124.224000,"
  [1342] = "-21.559000,-8.708000,137.357000,179.843000,0.299000,-124.623000,"
  [1343] = "-21.487000,-8.334000,137.364000,179.847000,0.294000,-124.996000,"
  [1344] = "-21.426000,-7.977000,137.370000,179.851000,0.289000,-125.331000,"
  [1345] = "-21.369000,-7.595000,137.376000,179.854000,0.285000,-125.665000,"
  [1346] = "-21.327000,-7.281000,137.381000,179.856000,0.282000,-125.924000,"
  [1347] = "-21.290000,-6.974000,137.386000,179.858000,0.280000,-126.165000,"
  [1348] = "-21.231000,-6.634000,137.392000,179.862000,0.274000,-126.520000,"
  [1349] = "-21.143000,-6.303000,137.400000,179.869000,0.262000,-127.029000,"
  [1350] = "-21.063000,-6.078000,137.407000,179.876000,0.251000,-127.500000,"
  [1351] = "-20.956000,-5.841000,137.416000,179.886000,0.235000,-128.144000,"
  [1352] = "-20.846000,-5.646000,137.424000,179.895000,0.220000,-128.839000,"
  [1353] = "-20.714000,-5.465000,137.434000,179.905000,0.202000,-129.709000,"
  [1354] = "-20.580000,-5.329000,137.443000,179.916000,0.183000,-130.624000,"
  [1355] = "-20.412000,-5.209000,137.454000,179.929000,0.160000,-131.800000,"
  [1356] = "-20.238000,-5.130000,137.465000,179.941000,0.135000,-133.042000,"
  [1357] = "-20.038000,-5.079000,137.477000,179.955000,0.107000,-134.489000,"
  [1358] = "-19.840000,-5.030000,137.488000,179.967000,0.081000,-135.995000,"
  [1359] = "-19.654000,-4.971000,137.499000,179.977000,0.059000,-137.491000,"
  [1360] = "-19.523000,-4.920000,137.506000,179.983000,0.044000,-138.613000,"
  [1361] = "-19.356000,-4.845000,137.515000,179.990000,0.029000,-140.122000,"
  [1362] = "-19.201000,-4.763000,137.522000,179.994000,0.017000,-141.614000,"
  [1363] = "-19.075000,-4.687000,137.529000,179.997000,0.008000,-142.904000,"
  [1364] = "-18.966000,-4.616000,137.534000,179.999000,0.003000,-144.073000,"
  [1365] = "-18.825000,-4.514000,137.540000,-179.999000,-0.003000,-145.667000,"
  [1366] = "-18.699000,-4.415000,137.546000,-179.998000,-0.006000,-147.184000,"
  [1367] = "-18.584000,-4.317000,137.550000,-179.998000,-0.008000,-148.636000,"
  [1368] = "-18.479000,-4.221000,137.555000,-179.998000,-0.009000,-150.028000,"
  [1369] = "-18.384000,-4.125000,137.558000,-179.998000,-0.008000,-151.368000,"
  [1370] = "-18.296000,-4.031000,137.562000,-179.999000,-0.006000,-152.663000,"
  [1371] = "-18.217000,-3.938000,137.564000,-179.999000,-0.003000,-153.918000,"
  [1372] = "-18.143000,-3.846000,137.567000,180.000000,0.001000,-155.138000,"
  [1373] = "-18.076000,-3.756000,137.569000,179.999000,0.006000,-156.327000,"
  [1374] = "-18.015000,-3.667000,137.570000,179.998000,0.012000,-157.489000,"
  [1375] = "-17.935000,-3.540000,137.572000,179.996000,0.022000,-159.140000,"
  [1376] = "-17.874000,-3.432000,137.573000,179.994000,0.032000,-160.544000,"
  [1377] = "-17.820000,-3.327000,137.574000,179.993000,0.043000,-161.908000,"
  [1378] = "-17.765000,-3.206000,137.574000,179.992000,0.058000,-163.482000,"
  [1379] = "-17.717000,-3.090000,137.574000,179.990000,0.074000,-165.047000,"
  [1380] = "-17.675000,-2.979000,137.573000,179.989000,0.091000,-166.582000,"
  [1381] = "-17.639000,-2.875000,137.572000,179.989000,0.108000,-168.101000,"
  [1382] = "-17.607000,-2.776000,137.571000,179.988000,0.127000,-169.605000,"
  [1383] = "-17.580000,-2.682000,137.569000,179.989000,0.145000,-171.097000,"
  [1384] = "-17.556000,-2.594000,137.567000,179.989000,0.164000,-172.581000,"
  [1385] = "-17.535000,-2.512000,137.565000,179.991000,0.183000,-174.058000,"
  [1386] = "-17.517000,-2.435000,137.563000,179.992000,0.202000,-175.529000,"
  [1387] = "-17.500000,-2.363000,137.560000,179.994000,0.221000,-176.997000,"
  [1388] = "-17.486000,-2.296000,137.558000,179.997000,0.240000,-178.461000,"
  [1389] = "-17.475000,-2.208000,137.554000,-179.999000,0.266000,179.622000,"
  [1390] = "-17.472000,-2.117000,137.549000,-179.994000,0.295000,177.754000,"
  [1391] = "-17.478000,-2.026000,137.544000,-179.988000,0.324000,175.928000,"
  [1392] = "-17.493000,-1.935000,137.538000,-179.982000,0.356000,174.139000,"
  [1393] = "-17.515000,-1.842000,137.532000,-179.974000,0.388000,172.388000,"
  [1394] = "-17.547000,-1.743000,137.525000,-179.966000,0.423000,170.696000,"
  [1395] = "-17.585000,-1.639000,137.518000,-179.956000,0.458000,169.059000,"
  [1396] = "-17.628000,-1.530000,137.511000,-179.946000,0.492000,167.472000,"
  [1397] = "-17.672000,-1.415000,137.504000,-179.935000,0.526000,165.930000,"
  [1398] = "-17.716000,-1.296000,137.497000,-179.924000,0.557000,164.428000,"
  [1399] = "-17.760000,-1.173000,137.490000,-179.912000,0.587000,162.962000,"
  [1400] = "-17.805000,-1.046000,137.484000,-179.900000,0.615000,161.530000,"
  [1401] = "-17.852000,-0.915000,137.477000,-179.888000,0.641000,160.130000,"
  [1402] = "-17.902000,-0.780000,137.471000,-179.875000,0.668000,158.760000,"
  [1403] = "-17.956000,-0.641000,137.464000,-179.861000,0.694000,157.419000,"
  [1404] = "-18.015000,-0.500000,137.457000,-179.847000,0.721000,156.105000,"
  [1405] = "-18.079000,-0.356000,137.450000,-179.833000,0.748000,154.817000,"
  [1406] = "-18.150000,-0.210000,137.443000,-179.818000,0.776000,153.551000,"
  [1407] = "-18.228000,-0.062000,137.435000,-179.801000,0.806000,152.308000,"
  [1408] = "-18.313000,0.084000,137.427000,-179.784000,0.837000,151.073000,"
  [1409] = "-18.403000,0.228000,137.419000,-179.766000,0.868000,149.833000,"
  [1410] = "-18.498000,0.367000,137.410000,-179.747000,0.900000,148.587000,"
  [1411] = "-18.598000,0.503000,137.401000,-179.727000,0.932000,147.332000,"
  [1412] = "-18.701000,0.635000,137.392000,-179.706000,0.963000,146.068000,"
  [1413] = "-18.807000,0.763000,137.383000,-179.685000,0.994000,144.794000,"
  [1414] = "-18.915000,0.887000,137.374000,-179.662000,1.024000,143.506000,"
  [1415] = "-19.026000,1.008000,137.365000,-179.639000,1.053000,142.205000,"
  [1416] = "-19.137000,1.124000,137.357000,-179.616000,1.081000,140.889000,"
  [1417] = "-19.249000,1.237000,137.348000,-179.592000,1.107000,139.555000,"
  [1418] = "-19.363000,1.354000,137.340000,-179.568000,1.133000,138.239000,"
  [1419] = "-19.421000,1.416000,137.335000,-179.556000,1.146000,137.600000,"
  [1420] = "-19.510000,1.514000,137.329000,-179.537000,1.165000,136.666000,"
  [1421] = "-19.631000,1.655000,137.320000,-179.512000,1.192000,135.467000,"
  [1422] = "-19.755000,1.807000,137.311000,-179.486000,1.219000,134.320000,"
  [1423] = "-19.881000,1.971000,137.302000,-179.461000,1.247000,133.226000,"
  [1424] = "-20.010000,2.147000,137.293000,-179.435000,1.275000,132.185000,"
  [1425] = "-20.141000,2.336000,137.284000,-179.409000,1.304000,131.198000,"
  [1426] = "-20.273000,2.537000,137.275000,-179.382000,1.332000,130.265000,"
  [1427] = "-20.407000,2.752000,137.266000,-179.356000,1.362000,129.386000,"
  [1428] = "-20.540000,2.977000,137.257000,-179.330000,1.390000,128.546000,"
  [1429] = "-20.674000,3.204000,137.249000,-179.304000,1.417000,127.703000,"
  [1430] = "-20.808000,3.432000,137.241000,-179.279000,1.442000,126.855000,"
  [1431] = "-20.942000,3.661000,137.234000,-179.254000,1.465000,126.001000,"
  [1432] = "-21.078000,3.892000,137.226000,-179.228000,1.487000,125.140000,"
  [1433] = "-21.215000,4.124000,137.220000,-179.203000,1.507000,124.272000,"
  [1434] = "-21.354000,4.357000,137.213000,-179.179000,1.525000,123.397000,"
  [1435] = "-21.496000,4.590000,137.207000,-179.154000,1.543000,122.515000,"
  [1436] = "-21.604000,4.766000,137.202000,-179.135000,1.555000,121.847000,"
  [1437] = "-21.742000,4.989000,137.197000,-179.112000,1.570000,121.005000,"
  [1438] = "-21.885000,5.231000,137.191000,-179.087000,1.586000,120.185000,"
  [1439] = "-22.007000,5.452000,137.186000,-179.067000,1.602000,119.531000,"
  [1440] = "-22.108000,5.646000,137.182000,-179.049000,1.615000,119.021000,"
  [1441] = "-22.246000,5.933000,137.177000,-179.025000,1.633000,118.362000,"
  [1442] = "-22.361000,6.195000,137.173000,-179.005000,1.650000,117.850000,"
  [1443] = "-22.450000,6.415000,137.169000,-178.990000,1.664000,117.476000,"
  [1444] = "-22.557000,6.703000,137.166000,-178.971000,1.681000,117.055000,"
  [1445] = "-22.639000,6.945000,137.163000,-178.957000,1.694000,116.754000,"
  [1446] = "-22.734000,7.263000,137.160000,-178.939000,1.711000,116.425000,"
  [1447] = "-22.804000,7.529000,137.158000,-178.927000,1.724000,116.200000,"
  [1448] = "-22.886000,7.872000,137.156000,-178.912000,1.740000,115.946000,"
  [1449] = "-22.949000,8.150000,137.156000,-178.901000,1.750000,115.747000,"
  [1450] = "-23.024000,8.502000,137.155000,-178.888000,1.762000,115.501000,"
  [1451] = "-23.082000,8.787000,137.154000,-178.879000,1.770000,115.308000,"
  [1452] = "-23.152000,9.148000,137.155000,-178.868000,1.779000,115.070000,"
  [1453] = "-23.206000,9.439000,137.155000,-178.860000,1.786000,114.884000,"
  [1454] = "-23.273000,9.806000,137.155000,-178.850000,1.793000,114.655000,"
  [1455] = "-23.326000,10.102000,137.156000,-178.843000,1.799000,114.475000,"
  [1456] = "-23.392000,10.475000,137.157000,-178.833000,1.805000,114.255000,"
  [1457] = "-23.444000,10.776000,137.158000,-178.826000,1.810000,114.082000,"
  [1458] = "-23.511000,11.153000,137.159000,-178.817000,1.817000,113.871000,"
  [1459] = "-23.565000,11.455000,137.160000,-178.810000,1.822000,113.703000,"
  [1460] = "-23.635000,11.834000,137.161000,-178.801000,1.829000,113.492000,"
  [1461] = "-23.693000,12.137000,137.162000,-178.793000,1.835000,113.323000,"
  [1462] = "-23.766000,12.516000,137.163000,-178.783000,1.842000,113.111000,"
  [1463] = "-23.826000,12.821000,137.164000,-178.776000,1.848000,112.940000,"
  [1464] = "-23.903000,13.201000,137.166000,-178.766000,1.855000,112.727000,"
  [1465] = "-23.965000,13.507000,137.167000,-178.758000,1.861000,112.555000,"
  [1466] = "-24.045000,13.889000,137.169000,-178.748000,1.868000,112.340000,"
  [1467] = "-24.110000,14.195000,137.170000,-178.740000,1.873000,112.167000,"
  [1468] = "-24.192000,14.580000,137.172000,-178.731000,1.880000,111.950000,"
  [1469] = "-24.258000,14.888000,137.173000,-178.723000,1.885000,111.776000,"
  [1470] = "-24.342000,15.274000,137.175000,-178.713000,1.891000,111.557000,"
  [1471] = "-24.410000,15.584000,137.176000,-178.706000,1.896000,111.382000,"
  [1472] = "-24.496000,15.974000,137.179000,-178.697000,1.902000,111.161000,"
  [1473] = "-24.565000,16.286000,137.180000,-178.690000,1.906000,110.985000,"
  [1474] = "-24.652000,16.678000,137.183000,-178.681000,1.910000,110.762000,"
  [1475] = "-24.722000,16.993000,137.185000,-178.675000,1.914000,110.584000,"
  [1476] = "-24.809000,17.388000,137.187000,-178.667000,1.917000,110.360000,"
  [1477] = "-24.880000,17.706000,137.189000,-178.661000,1.919000,110.180000,"
  [1478] = "-24.968000,18.106000,137.192000,-178.654000,1.921000,109.954000,"
  [1479] = "-25.038000,18.427000,137.195000,-178.648000,1.922000,109.773000,"
  [1480] = "-25.128000,18.829000,137.198000,-178.642000,1.923000,109.542000,"
  [1481] = "-25.200000,19.152000,137.200000,-178.637000,1.923000,109.355000,"
  [1482] = "-25.293000,19.556000,137.203000,-178.632000,1.922000,109.117000,"
  [1483] = "-25.370000,19.879000,137.206000,-178.627000,1.922000,108.924000,"
  [1484] = "-25.470000,20.283000,137.209000,-178.621000,1.922000,108.679000,"
  [1485] = "-25.553000,20.605000,137.211000,-178.616000,1.922000,108.479000,"
  [1486] = "-25.662000,21.007000,137.214000,-178.608000,1.923000,108.226000,"
  [1487] = "-25.753000,21.327000,137.217000,-178.602000,1.925000,108.020000,"
  [1488] = "-25.874000,21.725000,137.219000,-178.593000,1.928000,107.758000,"
  [1489] = "-25.975000,22.042000,137.221000,-178.585000,1.932000,107.550000,"
  [1490] = "-26.094000,22.447000,137.224000,-178.574000,1.938000,107.318000,"
  [1491] = "-26.198000,22.850000,137.228000,-178.564000,1.945000,107.127000,"
  [1492] = "-26.276000,23.208000,137.231000,-178.556000,1.951000,106.991000,"
  [1493] = "-26.349000,23.637000,137.235000,-178.548000,1.957000,106.865000,"
  [1494] = "-26.395000,24.021000,137.240000,-178.543000,1.961000,106.784000,"
  [1495] = "-26.426000,24.484000,137.245000,-178.541000,1.961000,106.722000,"
  [1496] = "-26.431000,24.900000,137.251000,-178.543000,1.958000,106.697000,"
  [1497] = "-26.408000,25.404000,137.257000,-178.550000,1.949000,106.700000,"
  [1498] = "-26.470000,25.781000,137.261000,-178.558000,1.931000,106.496000,"
  [1499] = "-26.460000,25.786000,137.678000,-178.559000,1.931000,106.513000,"
tool tTool = {fatherId=flange[0], ioLink=valve1}

--- start.pgx ---
program start()
begin
  call initdata()
  waitEndMove()
  delay(0)
  taskCreate "RobotMotion",100,RobotMotion()
  taskCreate "CmdTxtReading",85,CmdTxtReading()
  //  taskCreateSync "CmdTxtReading",0.004,btrig,CmdTxtReading()

  taskCreateSync "PositionTrigger",0.01,btrig,PositionTrigger()
end

--- CmdTxtReading.pgx ---
program CmdTxtReading()
begin
  while true
    if nTxtTotal>2
      if bTxt1==true
        call WipeCacheRoom1()
        delay(0)

        call TxtReadRoom1()
      else
      endIf
      if bTxt2==true
        call WipeCacheRoom2()
        delay(0)

        call TxtReadRoom2()
      else
      endIf
      if bTxt3==true
        call WipeCacheRoom3()
        delay(0)

        call TxtReadRoom3()
      else
      endIf
      delay(0)
    else
    endIf
  endWhile

end

--- initdata.pgx ---
program initdata()
begin
  nTxtTotal=11
  nNumTotal=5031
  n_sTxt=0
  nNumrecord=0
  fout=true
  bSignal=false
  bTxt1=false
  bTxt2=false
  bTxt3=false
  btrig=true
  call Txt_initData()
  call txt_PkgInit()

  //clearBuffer(sSocketout)
  //sioSet(sSocketout,nByteOut)
end

--- PositionTrigger.pgx ---
program PositionTrigger()
  local num nhere
begin
  ntime=clock()
  nnnn=0
  shere=pfrmCad[0]
  call Transmission()
  delay(0)

  while true
    if bSignal==true
      //shere=here(tTool,FrmDraw)
      shere=here(tTool,world)
      fout=false
      delay(0)
      fout=true
      delay(0.005)
      call Transmission()
      delay(0)
      ndelay=clock()-ntime
      nnnn=nnnn+1
    endIf
    delay(0)

  endWhile
  ndelay=clock()-ntime
end

--- RobotMotion.pgx ---
program RobotMotion()
  local num nNummove
begin
  movej(pfrmCad[0],tTool,mNomSpeed)
  waitEndMove()
  bSignal=true
  nNummove=0

  do
    movej(pfrmCad[nNummove],tTool,mNomSpeed)
    nNumrecord=nNumrecord+1

    if nNummove==600
      bTxt1=true
    endIf
    if nNummove==1100
      bTxt2=true
    endIf
    if nNummove==100
      bTxt3=true
    endIf
    delay(0)
    if nNummove==1499
      nNummove=0
    else
      nNummove=nNummove+1
    endIf
  until nNumrecord==nNumTotal
  waitEndMove()
  bSignal=false
  taskKill("PositionTrigger")
  ndelay=clock()-ntime
end

--- stop.pgx ---
program stop()
begin

end

--- stringtopoint.pgx ---
program stringtopoint(string x_sString (dimensions=1), num x_nNum (dimensions=1))
  local bool l_btest
  local num l_nNum6
  local string l_s
  local num nA
  local num nB
  local num nC
  local num nX
  local num nY
  local num nZ
  local pointRx pChangeMid1
  local pointRx pChangeMid2
  local trsf tTrsf
begin
  l_s=x_sString
  l_s=toNum(l_s,nX,l_btest)
  l_s=toNum(l_s,nY,l_btest)
  l_s=toNum(l_s,nZ,l_btest)
  l_s=toNum(l_s,nA,l_btest)
  l_s=toNum(l_s,nB,l_btest)
  l_s=toNum(l_s,nC,l_btest)
  pfrmCad[x_nNum].trsf={nX,nY,nZ,nA,nB,nC}
  link(pfrmCad[x_nNum],FrmDraw)
end

--- Transmission.pgx ---
program Transmission()
  local num nByteOut[48]
begin
  nTranC[0]=shere[0].trsf.x
  nTranC[1]=shere[0].trsf.y
  nTranC[2]=shere[0].trsf.z
  nTranC[3]=shere[0].trsf.rx
  nTranC[4]=shere[0].trsf.ry
  nTranC[5]=shere[0].trsf.rz

  //toBinary(nTranC,6,"8.0b",nByteOut)
  //sioSet(sSocketout,nByteOut)
  l_sString=toString(".3",nTranC[0])+","+toString(".3",nTranC[1])+","+toString(".3",nTranC[2])+","
  //l_sString=l_sString+toString(".3",nTranC[3])+","+toString(".3",nTranC[4])+","+toString(".3",nTranC[5])
  sSocketout=l_sString

end

--- txt_PkgInit.pgx ---
program txt_PkgInit()
begin
  call TxtReadRoom1()
  if nTxtTotal>1
    call TxtReadRoom2()
  endIf
end

--- TxtReadRoom1.pgx ---
program TxtReadRoom1()
  local string l_str
  local num nNumpoint
  local num ntext
  local string sTxtfile
begin
  bTxt1=false
  delay(0)
  l_str=toString("1",n_sTxt)
  sTxtfile="path"+l_str+".txt"
  ntext=$fileOpen(sTxtfile,"r")
  for nNumpoint=0 to 499
    $fileGet(ntext,sString[nNumpoint],1)
    if sString[nNumpoint]!=""
      call stringtopoint(sString[nNumpoint],nNumpoint)
    else
    endIf
  endFor
  delay(0)


  if n_sTxt==nTxtTotal-1
    n_sTxt=0
  elseIf n_sTxt!=nTxtTotal-1
    n_sTxt=n_sTxt+1
  endIf

  nNumpoint=nNumpoint-1
  $fileClose(ntext)
end

--- WipeCacheRoom3.pgx ---
program WipeCacheRoom3()
  local num nNum
begin
  for nNum=1000 to 1499
    sString[nNum]=""
    pfrmCad[nNum].trsf={0,0,0,0,0,0}
  endFor

end
